Staubli VAL3: VelocityCmdMsg.pjx

--- VelocityCmdMsg.pjx ---
Parameters version=s7.8.1 stackSize=5000 millimeterUnit=true
Program file=start.pgx
Program file=stop.pgx
Data file=VelocityCmdMsg.dtx
Type name=Body path=Disk://ros_libs/Body/Body.pjx
Type name=Prefix path=Disk://ros_libs/Prefix/Prefix.pjx
Type name=Header path=Disk://ros_libs/Header/Header.pjx
Type name=VelocityCmd path=../VelocityCmd/VelocityCmd.pjx

--- VelocityCmdMsg.dtx ---
public Header header
  [0]
    num nMsgType
    num nCommType
    num nReplyCode
    num nData[12]
public Body body
  [0]
    num nData[32]
public Prefix prefix
  [0]
    num nLength
    num nData[4]
public VelocityCmd velCmd
  [0]
    num nSeq
    num nVelVec[6]
    num nCmdType
